TYPE TcoInsightAcquisitionControl_v_5_x_x :
STRUCT
	AcquisitionTriggerEnable AT %Q* :  BOOL;
	AcquisitionTrigger AT %Q* :  BOOL;
	ClearExposureComplete AT %Q* :  BOOL;
	SetOffline AT %Q* :  BOOL;
END_STRUCT
END_TYPE

(* stored: Version 1.1.0.1, ProductVersion 3.1.4024.11
   DUT TcoInsightAcquisitionControl_v_5_x_x: Id {1768b1d4-1d86-032c-38d5-fb5c1542f51f} *)
